PROGRAM P_Demo_FB_PN_SCAN_UpTo255
VAR
    fbScan255     : FB_PN_SCAN_UpTo255;
    bScanReq      : BOOL := FALSE;            // 在线上升沿触发扫描
    bBusy         : BOOL;
    bErr          : BOOL;
    nErrId        : UDINT;
    iFound        : INT;                      // 扫描到的设备数
    aDevices      : ARRAY [1..255] OF str_PN_SCAN;   // 逐台设备信息（最多 255）
END_VAR

// ============================================================
// Tc2_ProfinetDiag.FB_PN_SCAN_UpTo255 演示程序
// ============================================================
// 场景：扫描全网 PROFINET 设备（≤255 台）。
// 价值：大网络一次扫全，免分批。
// 验证：登录后 bScanReq 上升沿，iFound/aDevices 填入（需库≥v1.5.2.0）。
// 验证步骤：
//   1. 右键 PLC 项目下 POUs 文件夹 → Add → Existing Item → 选本 .TcPOU 文件
//   2. 引用 Tc2_ProfinetDiag（References → Add library）
//   3. 编译 → 登录 → 运行；按上方『验证』指引在线写值观察
// ============================================================

// 上升沿触发；扫描全网（最多 255 台，需库 >= v1.5.2.0）
fbScan255(
    bExecute := bScanReq,
    NETID    := '',
    iFind_Devices => iFound,
    ar_PN_DEVICE => aDevices,
    bBusy    => bBusy,
    bError   => bErr,
    iErrorID => nErrId
);

END_PROGRAM

(* stored: Version 1.1.0.1, ProductVersion 3.1.4024.5
   POU P_Demo_FB_PN_SCAN_UpTo255: Id {0bcfdf31-280c-523f-acdb-272fb22e718f}, SpecialFunc None *)
